VAR_GLOBAL
END_VAR

(* stored: Version 1.1.0.1, ProductVersion 3.1.0.25
   GVL POD_Const: Id {3db20bdd-54f7-4841-b871-6cc1b7237e45} *)
